// TIA Portal project "COUNTER_1_3" (V14)

(* hardware
DEVICE "S7-1200 station_1"  S7-1200 Station
   slot 0: "Rack_0"  S7-1200 Rack  Rack  V1.0
   slot 1: "CPU"  CPU 1212C DC/DC/DC  6ES7 212-1AE40-0XB0  V4.2
DEVICE "HMI_1"  KTP400 Basic PN
   slot 0: "KTP400 Basic PN"  KTP400 Basic PN  6AV2 123-2DB03-0AX0  14.0.1.0
   slot 1: "HMI_RT_1"  KTP400 Basic PN  6AV2 123-2DB03-0AX0  14.0.1.0
   slot 5: "HMI_1.IE_CP_1"  PROFINET Interface  14.0.1.0
      slot 1: "PROFINET Interface_1"  PROFINET Interface
         slot 1: "Port_1"  Port
DEVICE "HMI_2"  KTP400 Basic PN
   slot 0: "KTP400 Basic PN"  KTP400 Basic PN  6AV2 123-2DB03-0AX0  14.0.1.0
   slot 1: "HMI_RT_2"  KTP400 Basic PN  6AV2 123-2DB03-0AX0  14.0.1.0
   slot 5: "HMI_1.IE_CP_1"  PROFINET Interface  14.0.1.0
      slot 1: "PROFINET Interface_1"  PROFINET Interface
         slot 1: "Port_1"  Port
*)

// ===== PLC "CPU"  CPU 1212C DC/DC/DC =====

VAR_GLOBAL   // PLC tag table "Default tag table"
   "CNT_1_IMP" AT %ID1000 : DWord;
   "CNT_2_IMP" AT %ID1004 : DInt;
   "StopFromCNT_2" AT %Q0.0 : Bool;   // Стоп от счетчика метража машина 1
   "CNN_3_IMP" AT %ID1008 : DInt;
   "CNT_4_IMP" AT %ID1012 : DInt;
   "StopFromCNT_4" AT %Q0.1 : Bool;
   "Tag_1" AT %MW10 : Word;
   "Tag_2" AT %MD10 : Real;
   "Tag_3" AT %MD15 : Real;
END_VAR

DATA_BLOCK "DSE_1"   // DB3
{ S7_Optimized_Access := 'TRUE' }
VERSION : 0.1
   VAR RETAIN
      "Счетчик импульсов 1" : DInt;
      "Счетчик импульсов 2" : DInt;
   END_VAR
   VAR
      "Сброс счетчика 1" : Bool;
      "Сброс счетчика 2" : Bool;
   END_VAR
   VAR RETAIN
      "Диаметр колеса пасма" : Real := 0.106;
      "Количество импулсов на оборот пасма" : Real := 1.0;
      "Коэффициент счетчика пасма" : Real := 1.0;
      "Метраж пасма" : Real;
      "Коэффициент трансмиссии рамки" : Real := 1.0;
      "Шаг скрутки в метрах (выбранной ступени)" : Real;
      "Коэффициент метража жилы (выбранной ступени)" : Real := 1.0;
      "метраж жила" : Real;
      "Номер ступени" : Int;
      "Ступень 0 Шаг" : Real := 0.0091;
      "Ступень 1 Шаг" : Real := 0.0114;
      "Ступень 2 Шаг" : Real := 0.0141;
      "Ступень 3 Шаг" : Real := 0.0181;
      "Ступень 4 Шаг" : Real := 0.0228;
      "Ступень 5 Шаг" : Real := 0.0316;
      "Ступень 6 Шаг" : Real := 0.04;
      "Ступень 7 Шаг" : Real := 0.0511;
      "Ступень 8 Шаг" : Real := 0.0631;
      "Ступень 9 Шаг" : Real := 0.0794;
      "Ступень 10 Шаг" : Real := 0.091;
      "Метраж заданый" : Real;
      "Ступень 0 Коэффициент метража жилы" : Real := 0.9791;
      "Ступень 1 Коэффициент метража жилы" : Real := 0.9791;
      "Ступень 2 Коэффициент метража жилы" : Real := 0.9791;
      "Ступень 3 Коэффициент метража жилы" : Real := 0.9791;
      "Ступень 4 Коэффициент метража жилы" : Real := 0.9791;
      "Ступень 5 Коэффициент метража жилы" : Real := 0.9791;
      "Ступень 6 Коэффициент метража жилы" : Real := 0.9791;
      "Ступень 7 Коэффициент метража жилы" : Real := 0.9791;
      "Ступень 8 Коэффициент метража жилы" : Real := 0.9791;
      "Ступень 9 Коэффициент метража жилы" : Real := 0.9791;
      "Ступень 10 Коэффициент метража жилы" : Real := 0.9791;
   END_VAR
   VAR
      "Скорость DSE 1" : Real;
   END_VAR
BEGIN
END_DATA_BLOCK

DATA_BLOCK "DSE_3"   // DB6
{ S7_Optimized_Access := 'TRUE' }
VERSION : 0.1
   VAR RETAIN
      "Счетчик импульсов 1" : DInt;
      "Счетчик импульсов 2" : DInt;
   END_VAR
   VAR
      "Сброс счетчика 1" : Bool;
      "Сброс счетчика 2" : Bool;
   END_VAR
   VAR RETAIN
      "Диаметр колеса пасма" : Real := 0.106;
      "Количество импулсов на оборот пасма" : Real := 1.0;
      "Коэффициент счетчика пасма" : Real := 1.0;
      "Метраж пасма" : Real;
      "Коэффициент трансмиссии рамки" : Real := 1.0;
      "Шаг скрутки в метрах (выбранной ступени)" : Real;
      "Коэффициент метража жилы (выбранной ступени)" : Real := 1.0;
      "метраж жила" : Real;
      "Номер ступени" : Int;
      "Ступень 0 Шаг" : Real := 0.0091;
      "Ступень 1 Шаг" : Real := 0.0114;
      "Ступень 2 Шаг" : Real := 0.0141;
      "Ступень 3 Шаг" : Real := 0.0181;
      "Ступень 4 Шаг" : Real := 0.0228;
      "Ступень 5 Шаг" : Real := 0.0316;
      "Ступень 6 Шаг" : Real := 0.04;
      "Ступень 7 Шаг" : Real := 0.0511;
      "Ступень 8 Шаг" : Real := 0.0631;
      "Ступень 9 Шаг" : Real := 0.0794;
      "Ступень 10 Шаг" : Real := 0.091;
      "Метраж заданый" : Real;
      "Ступень 0 Коэффициент метража жилы" : Real := 0.9791;
      "Ступень 1 Коэффициент метража жилы" : Real := 0.9791;
      "Ступень 2 Коэффициент метража жилы" : Real := 0.9791;
      "Ступень 3 Коэффициент метража жилы" : Real := 0.9791;
      "Ступень 4 Коэффициент метража жилы" : Real := 0.9791;
      "Ступень 5 Коэффициент метража жилы" : Real := 0.9791;
      "Ступень 6 Коэффициент метража жилы" : Real := 0.9791;
      "Ступень 7 Коэффициент метража жилы" : Real := 0.9791;
      "Ступень 8 Коэффициент метража жилы" : Real := 0.9791;
      "Ступень 9 Коэффициент метража жилы" : Real := 0.9791;
      "Ступень 10 Коэффициент метража жилы" : Real := 0.9791;
   END_VAR
   VAR
      "Скорость DSE 1" : Real;
   END_VAR
BEGIN
END_DATA_BLOCK

ORGANIZATION_BLOCK "Main"   // OB1, LAD, ProgramCycle
TITLE = "Main Program Sweep (Cycle)"
{ S7_Optimized_Access := 'TRUE' }
VERSION : 0.1
   VAR_INPUT
      Initial_Call : Bool;   // Initial call of this OB
      Remanence : Bool;   // =True, if remanent data are available
   END_VAR
BEGIN

REGION Network 1: DSE 1
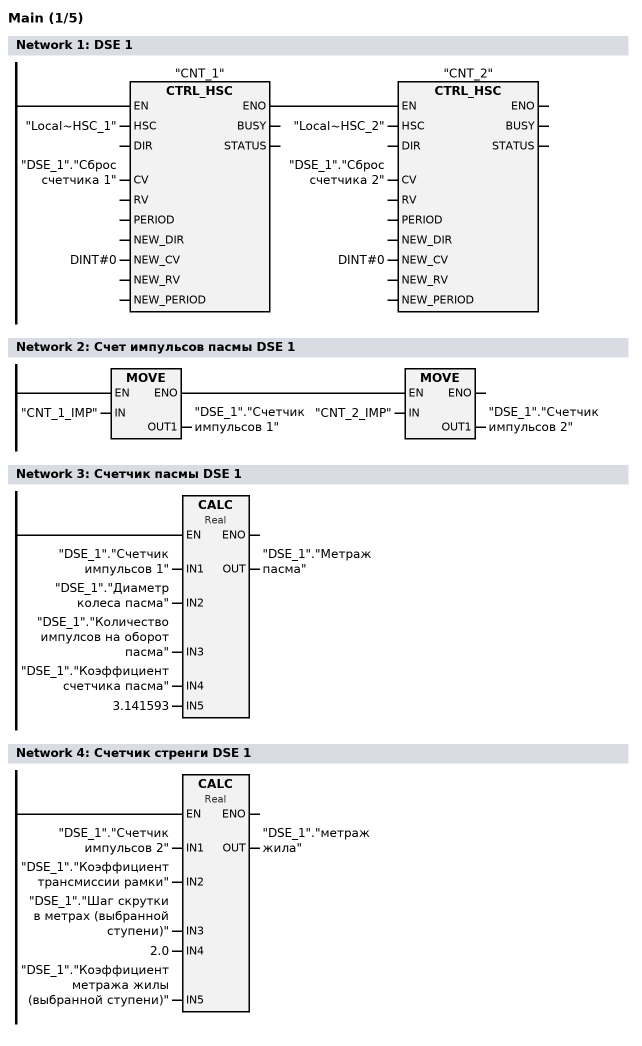
   // ENO of a box is taken as its EN; it also drops when the box reports an error
   "CNT_1"(HSC := "Local~HSC_1", CV := "DSE_1"."Сброс счетчика 1", NEW_CV := DINT#0);   // CTRL_HSC
   "CNT_2"(HSC := "Local~HSC_2", CV := "DSE_1"."Сброс счетчика 2", NEW_CV := DINT#0);   // CTRL_HSC
END_REGION

REGION Network 2: Счет импульсов пасмы DSE 1
   RUNG wire#powerrail
      Move(in := "CNT_1_IMP", out1 => "DSE_1"."Счетчик импульсов 1")
      Move(in := "CNT_2_IMP", out1 => "DSE_1"."Счетчик импульсов 2")
   END_RUNG
   // the same network as SCL:
   "DSE_1"."Счетчик импульсов 1" := "CNT_1_IMP";
   "DSE_1"."Счетчик импульсов 2" := "CNT_2_IMP";
END_REGION

REGION Network 3: Счетчик пасмы DSE 1
   CALC(in1 := "DSE_1"."Счетчик импульсов 1",
        in2 := "DSE_1"."Диаметр колеса пасма",
        in3 := "DSE_1"."Количество импулсов на оборот пасма",
        in4 := "DSE_1"."Коэффициент счетчика пасма",
        in5 := 3.141593,
        out => "DSE_1"."Метраж пасма");
END_REGION

REGION Network 4: Счетчик стренги DSE 1
   CALC(in1 := "DSE_1"."Счетчик импульсов 2",
        in2 := "DSE_1"."Коэффициент трансмиссии рамки",
        in3 := "DSE_1"."Шаг скрутки в метрах (выбранной ступени)",
        in4 := 2.0,
        in5 := "DSE_1"."Коэффициент метража жилы (выбранной ступени)",
        out => "DSE_1"."метраж жила");
END_REGION

REGION Network 5: Загрузка шага скрутки в метрах DSE 1
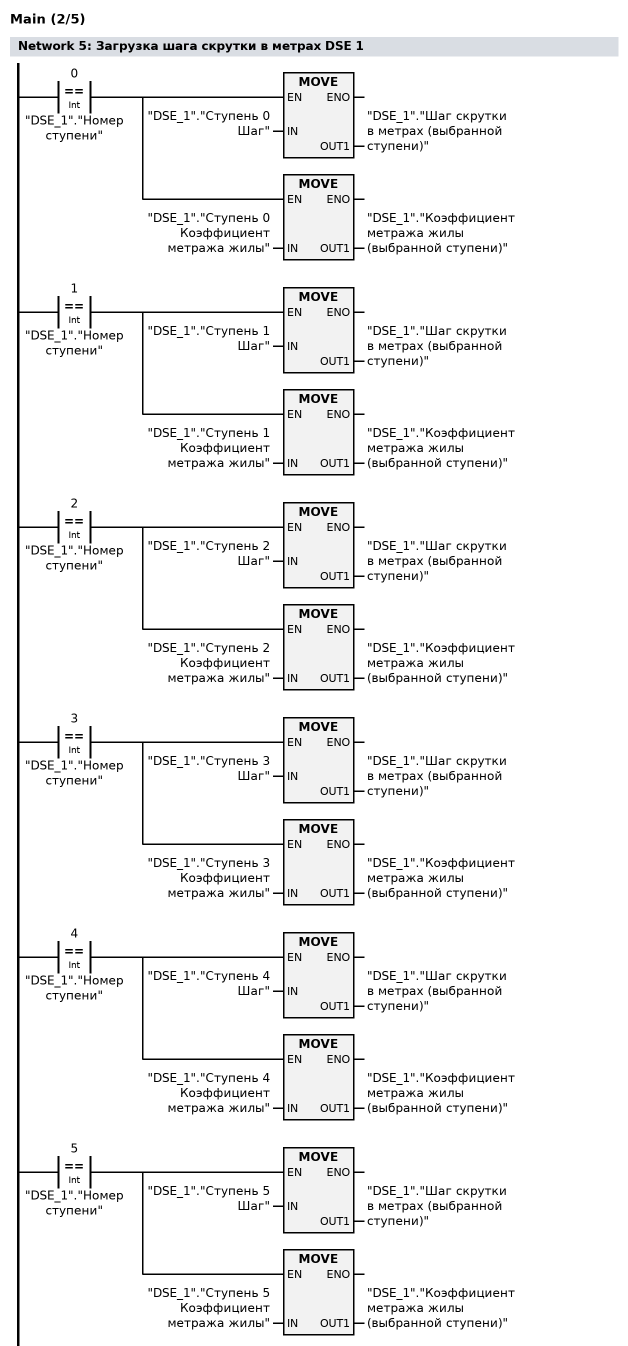
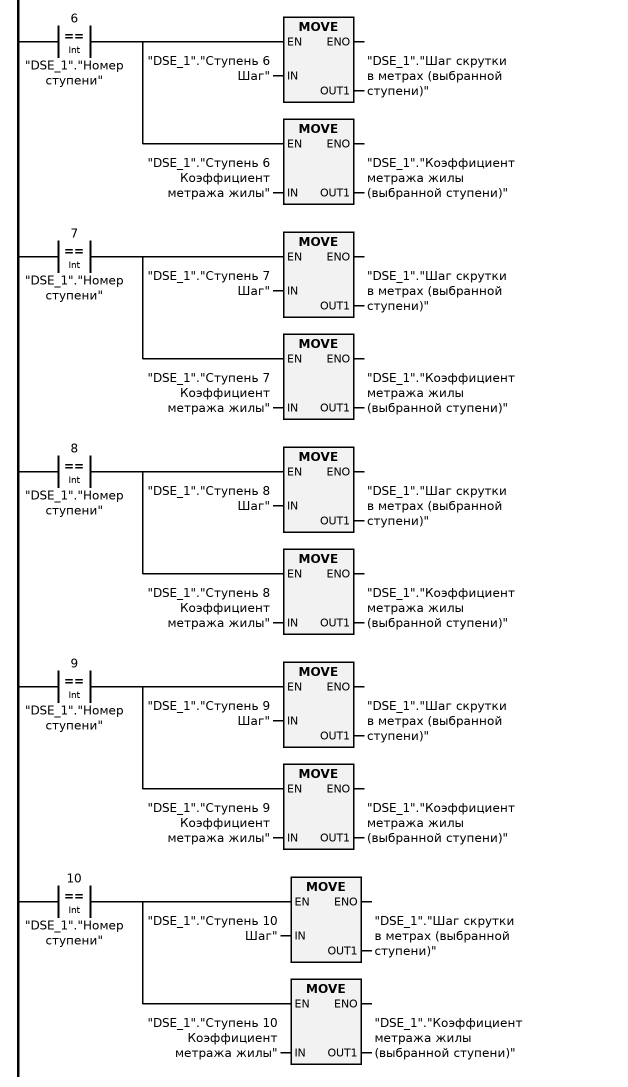
   RUNG wire#powerrail
      { S7_Templates := "SrcType := Int" } EQ_Contact(in1 := 0, in2 := "DSE_1"."Номер ступени")
      wire#w1
      Move(in := "DSE_1"."Ступень 0 Шаг", out1 => "DSE_1"."Шаг скрутки в метрах (выбранной ступени)")
   END_RUNG
   RUNG wire#w1
      Move(in := "DSE_1"."Ступень 0 Коэффициент метража жилы", out1 => "DSE_1"."Коэффициент метража жилы (выбранной ступени)")
   END_RUNG
   RUNG wire#powerrail
      { S7_Templates := "SrcType := Int" } EQ_Contact(in1 := 1, in2 := "DSE_1"."Номер ступени")
      wire#w2
      Move(in := "DSE_1"."Ступень 1 Шаг", out1 => "DSE_1"."Шаг скрутки в метрах (выбранной ступени)")
   END_RUNG
   RUNG wire#w2
      Move(in := "DSE_1"."Ступень 1 Коэффициент метража жилы", out1 => "DSE_1"."Коэффициент метража жилы (выбранной ступени)")
   END_RUNG
   RUNG wire#powerrail
      { S7_Templates := "SrcType := Int" } EQ_Contact(in1 := 2, in2 := "DSE_1"."Номер ступени")
      wire#w3
      Move(in := "DSE_1"."Ступень 2 Шаг", out1 => "DSE_1"."Шаг скрутки в метрах (выбранной ступени)")
   END_RUNG
   RUNG wire#w3
      Move(in := "DSE_1"."Ступень 2 Коэффициент метража жилы", out1 => "DSE_1"."Коэффициент метража жилы (выбранной ступени)")
   END_RUNG
   RUNG wire#powerrail
      { S7_Templates := "SrcType := Int" } EQ_Contact(in1 := 3, in2 := "DSE_1"."Номер ступени")
      wire#w4
      Move(in := "DSE_1"."Ступень 3 Шаг", out1 => "DSE_1"."Шаг скрутки в метрах (выбранной ступени)")
   END_RUNG
   RUNG wire#w4
      Move(in := "DSE_1"."Ступень 3 Коэффициент метража жилы", out1 => "DSE_1"."Коэффициент метража жилы (выбранной ступени)")
   END_RUNG
   RUNG wire#powerrail
      { S7_Templates := "SrcType := Int" } EQ_Contact(in1 := 4, in2 := "DSE_1"."Номер ступени")
      wire#w5
      Move(in := "DSE_1"."Ступень 4 Шаг", out1 => "DSE_1"."Шаг скрутки в метрах (выбранной ступени)")
   END_RUNG
   RUNG wire#w5
      Move(in := "DSE_1"."Ступень 4 Коэффициент метража жилы", out1 => "DSE_1"."Коэффициент метража жилы (выбранной ступени)")
   END_RUNG
   RUNG wire#powerrail
      { S7_Templates := "SrcType := Int" } EQ_Contact(in1 := 5, in2 := "DSE_1"."Номер ступени")
      wire#w6
      Move(in := "DSE_1"."Ступень 5 Шаг", out1 => "DSE_1"."Шаг скрутки в метрах (выбранной ступени)")
   END_RUNG
   RUNG wire#w6
      Move(in := "DSE_1"."Ступень 5 Коэффициент метража жилы", out1 => "DSE_1"."Коэффициент метража жилы (выбранной ступени)")
   END_RUNG
   RUNG wire#powerrail
      { S7_Templates := "SrcType := Int" } EQ_Contact(in1 := 6, in2 := "DSE_1"."Номер ступени")
      wire#w7
      Move(in := "DSE_1"."Ступень 6 Шаг", out1 => "DSE_1"."Шаг скрутки в метрах (выбранной ступени)")
   END_RUNG
   RUNG wire#w7
      Move(in := "DSE_1"."Ступень 6 Коэффициент метража жилы", out1 => "DSE_1"."Коэффициент метража жилы (выбранной ступени)")
   END_RUNG
   RUNG wire#powerrail
      { S7_Templates := "SrcType := Int" } EQ_Contact(in1 := 7, in2 := "DSE_1"."Номер ступени")
      wire#w8
      Move(in := "DSE_1"."Ступень 7 Шаг", out1 => "DSE_1"."Шаг скрутки в метрах (выбранной ступени)")
   END_RUNG
   RUNG wire#w8
      Move(in := "DSE_1"."Ступень 7 Коэффициент метража жилы", out1 => "DSE_1"."Коэффициент метража жилы (выбранной ступени)")
   END_RUNG
   RUNG wire#powerrail
      { S7_Templates := "SrcType := Int" } EQ_Contact(in1 := 8, in2 := "DSE_1"."Номер ступени")
      wire#w9
      Move(in := "DSE_1"."Ступень 8 Шаг", out1 => "DSE_1"."Шаг скрутки в метрах (выбранной ступени)")
   END_RUNG
   RUNG wire#w9
      Move(in := "DSE_1"."Ступень 8 Коэффициент метража жилы", out1 => "DSE_1"."Коэффициент метража жилы (выбранной ступени)")
   END_RUNG
   RUNG wire#powerrail
      { S7_Templates := "SrcType := Int" } EQ_Contact(in1 := 9, in2 := "DSE_1"."Номер ступени")
      wire#w10
      Move(in := "DSE_1"."Ступень 9 Шаг", out1 => "DSE_1"."Шаг скрутки в метрах (выбранной ступени)")
   END_RUNG
   RUNG wire#w10
      Move(in := "DSE_1"."Ступень 9 Коэффициент метража жилы", out1 => "DSE_1"."Коэффициент метража жилы (выбранной ступени)")
   END_RUNG
   RUNG wire#powerrail
      { S7_Templates := "SrcType := Int" } EQ_Contact(in1 := 10, in2 := "DSE_1"."Номер ступени")
      wire#w11
      Move(in := "DSE_1"."Ступень 10 Шаг", out1 => "DSE_1"."Шаг скрутки в метрах (выбранной ступени)")
   END_RUNG
   RUNG wire#w11
      Move(in := "DSE_1"."Ступень 10 Коэффициент метража жилы", out1 => "DSE_1"."Коэффициент метража жилы (выбранной ступени)")
   END_RUNG
   // the same network as SCL:
   IF 0 = "DSE_1"."Номер ступени" THEN
       "DSE_1"."Шаг скрутки в метрах (выбранной ступени)" := "DSE_1"."Ступень 0 Шаг";
       "DSE_1"."Коэффициент метража жилы (выбранной ступени)" := "DSE_1"."Ступень 0 Коэффициент метража жилы";
   END_IF;
   IF 1 = "DSE_1"."Номер ступени" THEN
       "DSE_1"."Шаг скрутки в метрах (выбранной ступени)" := "DSE_1"."Ступень 1 Шаг";
       "DSE_1"."Коэффициент метража жилы (выбранной ступени)" := "DSE_1"."Ступень 1 Коэффициент метража жилы";
   END_IF;
   IF 2 = "DSE_1"."Номер ступени" THEN
       "DSE_1"."Шаг скрутки в метрах (выбранной ступени)" := "DSE_1"."Ступень 2 Шаг";
       "DSE_1"."Коэффициент метража жилы (выбранной ступени)" := "DSE_1"."Ступень 2 Коэффициент метража жилы";
   END_IF;
   IF 3 = "DSE_1"."Номер ступени" THEN
       "DSE_1"."Шаг скрутки в метрах (выбранной ступени)" := "DSE_1"."Ступень 3 Шаг";
       "DSE_1"."Коэффициент метража жилы (выбранной ступени)" := "DSE_1"."Ступень 3 Коэффициент метража жилы";
   END_IF;
   IF 4 = "DSE_1"."Номер ступени" THEN
       "DSE_1"."Шаг скрутки в метрах (выбранной ступени)" := "DSE_1"."Ступень 4 Шаг";
       "DSE_1"."Коэффициент метража жилы (выбранной ступени)" := "DSE_1"."Ступень 4 Коэффициент метража жилы";
   END_IF;
   IF 5 = "DSE_1"."Номер ступени" THEN
       "DSE_1"."Шаг скрутки в метрах (выбранной ступени)" := "DSE_1"."Ступень 5 Шаг";
       "DSE_1"."Коэффициент метража жилы (выбранной ступени)" := "DSE_1"."Ступень 5 Коэффициент метража жилы";
   END_IF;
   IF 6 = "DSE_1"."Номер ступени" THEN
       "DSE_1"."Шаг скрутки в метрах (выбранной ступени)" := "DSE_1"."Ступень 6 Шаг";
       "DSE_1"."Коэффициент метража жилы (выбранной ступени)" := "DSE_1"."Ступень 6 Коэффициент метража жилы";
   END_IF;
   IF 7 = "DSE_1"."Номер ступени" THEN
       "DSE_1"."Шаг скрутки в метрах (выбранной ступени)" := "DSE_1"."Ступень 7 Шаг";
       "DSE_1"."Коэффициент метража жилы (выбранной ступени)" := "DSE_1"."Ступень 7 Коэффициент метража жилы";
   END_IF;
   IF 8 = "DSE_1"."Номер ступени" THEN
       "DSE_1"."Шаг скрутки в метрах (выбранной ступени)" := "DSE_1"."Ступень 8 Шаг";
       "DSE_1"."Коэффициент метража жилы (выбранной ступени)" := "DSE_1"."Ступень 8 Коэффициент метража жилы";
   END_IF;
   IF 9 = "DSE_1"."Номер ступени" THEN
       "DSE_1"."Шаг скрутки в метрах (выбранной ступени)" := "DSE_1"."Ступень 9 Шаг";
       "DSE_1"."Коэффициент метража жилы (выбранной ступени)" := "DSE_1"."Ступень 9 Коэффициент метража жилы";
   END_IF;
   IF 10 = "DSE_1"."Номер ступени" THEN
       "DSE_1"."Шаг скрутки в метрах (выбранной ступени)" := "DSE_1"."Ступень 10 Шаг";
       "DSE_1"."Коэффициент метража жилы (выбранной ступени)" := "DSE_1"."Ступень 10 Коэффициент метража жилы";
   END_IF;
END_REGION

REGION Network 6: Стоп по счетчику DSE 1
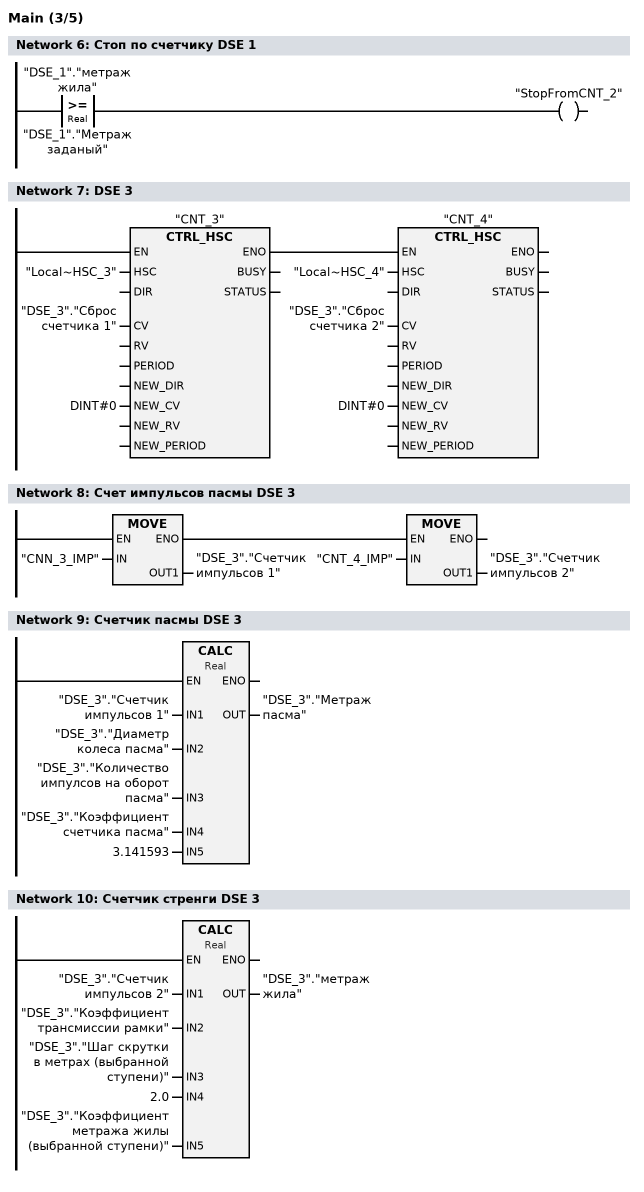
   RUNG wire#powerrail
      { S7_Templates := "SrcType := Real" } GE_Contact(in1 := "DSE_1"."метраж жила", in2 := "DSE_1"."Метраж заданый")
      Coil( "StopFromCNT_2" )
   END_RUNG
   // the same network as SCL:
   "StopFromCNT_2" := "DSE_1"."метраж жила" >= "DSE_1"."Метраж заданый";
END_REGION

REGION Network 7: DSE 3
   // ENO of a box is taken as its EN; it also drops when the box reports an error
   "CNT_3"(HSC := "Local~HSC_3", CV := "DSE_3"."Сброс счетчика 1", NEW_CV := DINT#0);   // CTRL_HSC
   "CNT_4"(HSC := "Local~HSC_4", CV := "DSE_3"."Сброс счетчика 2", NEW_CV := DINT#0);   // CTRL_HSC
END_REGION

REGION Network 8: Счет импульсов пасмы DSE 3
   RUNG wire#powerrail
      Move(in := "CNN_3_IMP", out1 => "DSE_3"."Счетчик импульсов 1")
      Move(in := "CNT_4_IMP", out1 => "DSE_3"."Счетчик импульсов 2")
   END_RUNG
   // the same network as SCL:
   "DSE_3"."Счетчик импульсов 1" := "CNN_3_IMP";
   "DSE_3"."Счетчик импульсов 2" := "CNT_4_IMP";
END_REGION

REGION Network 9: Счетчик пасмы DSE 3
   CALC(in1 := "DSE_3"."Счетчик импульсов 1",
        in2 := "DSE_3"."Диаметр колеса пасма",
        in3 := "DSE_3"."Количество импулсов на оборот пасма",
        in4 := "DSE_3"."Коэффициент счетчика пасма",
        in5 := 3.141593,
        out => "DSE_3"."Метраж пасма");
END_REGION

REGION Network 10: Счетчик стренги DSE 3
   CALC(in1 := "DSE_3"."Счетчик импульсов 2",
        in2 := "DSE_3"."Коэффициент трансмиссии рамки",
        in3 := "DSE_3"."Шаг скрутки в метрах (выбранной ступени)",
        in4 := 2.0,
        in5 := "DSE_3"."Коэффициент метража жилы (выбранной ступени)",
        out => "DSE_3"."метраж жила");
END_REGION

REGION Network 11: Загрузка шага скрутки в метрах DSE 3
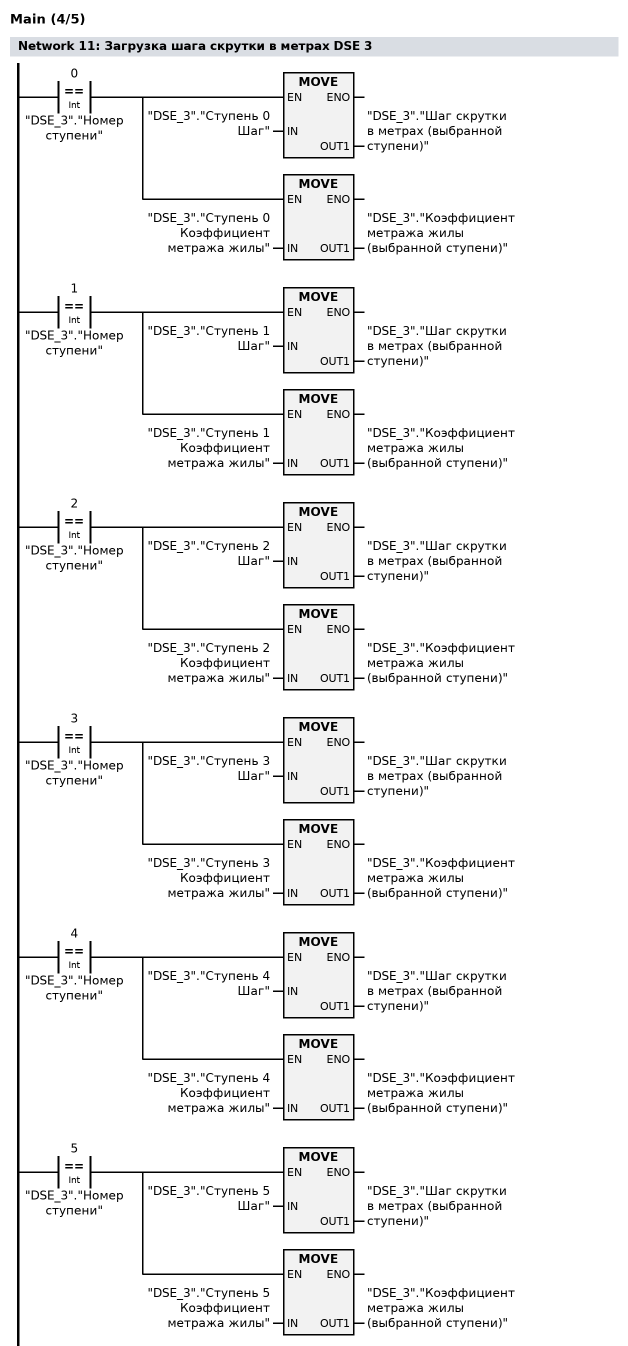
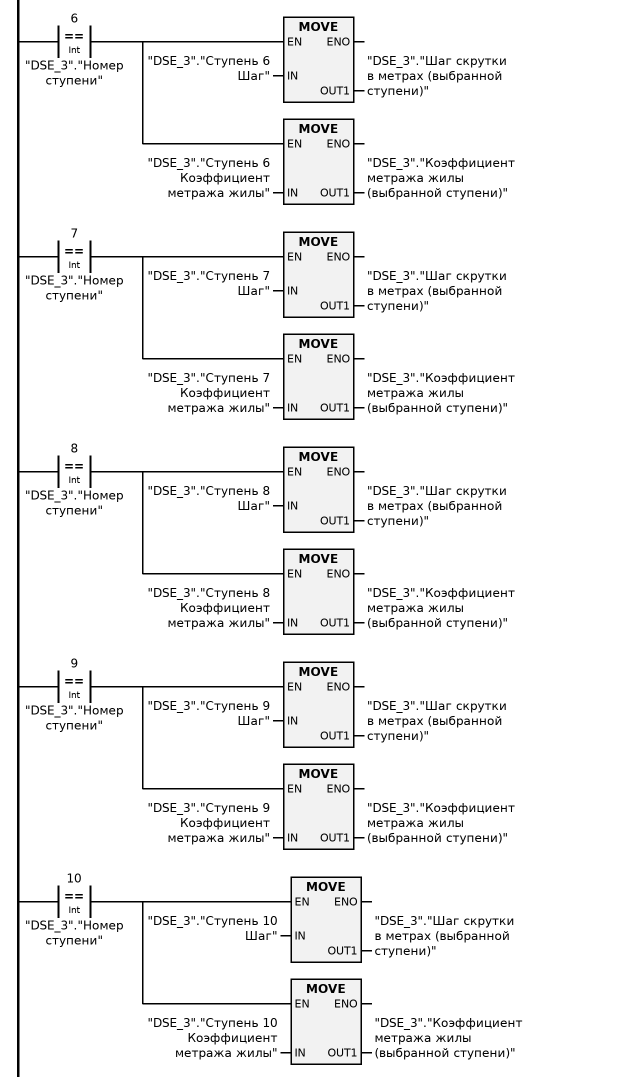
   RUNG wire#powerrail
      { S7_Templates := "SrcType := Int" } EQ_Contact(in1 := 0, in2 := "DSE_3"."Номер ступени")
      wire#w1
      Move(in := "DSE_3"."Ступень 0 Шаг", out1 => "DSE_3"."Шаг скрутки в метрах (выбранной ступени)")
   END_RUNG
   RUNG wire#w1
      Move(in := "DSE_3"."Ступень 0 Коэффициент метража жилы", out1 => "DSE_3"."Коэффициент метража жилы (выбранной ступени)")
   END_RUNG
   RUNG wire#powerrail
      { S7_Templates := "SrcType := Int" } EQ_Contact(in1 := 1, in2 := "DSE_3"."Номер ступени")
      wire#w2
      Move(in := "DSE_3"."Ступень 1 Шаг", out1 => "DSE_3"."Шаг скрутки в метрах (выбранной ступени)")
   END_RUNG
   RUNG wire#w2
      Move(in := "DSE_3"."Ступень 1 Коэффициент метража жилы", out1 => "DSE_3"."Коэффициент метража жилы (выбранной ступени)")
   END_RUNG
   RUNG wire#powerrail
      { S7_Templates := "SrcType := Int" } EQ_Contact(in1 := 2, in2 := "DSE_3"."Номер ступени")
      wire#w3
      Move(in := "DSE_3"."Ступень 2 Шаг", out1 => "DSE_3"."Шаг скрутки в метрах (выбранной ступени)")
   END_RUNG
   RUNG wire#w3
      Move(in := "DSE_3"."Ступень 2 Коэффициент метража жилы", out1 => "DSE_3"."Коэффициент метража жилы (выбранной ступени)")
   END_RUNG
   RUNG wire#powerrail
      { S7_Templates := "SrcType := Int" } EQ_Contact(in1 := 3, in2 := "DSE_3"."Номер ступени")
      wire#w4
      Move(in := "DSE_3"."Ступень 3 Шаг", out1 => "DSE_3"."Шаг скрутки в метрах (выбранной ступени)")
   END_RUNG
   RUNG wire#w4
      Move(in := "DSE_3"."Ступень 3 Коэффициент метража жилы", out1 => "DSE_3"."Коэффициент метража жилы (выбранной ступени)")
   END_RUNG
   RUNG wire#powerrail
      { S7_Templates := "SrcType := Int" } EQ_Contact(in1 := 4, in2 := "DSE_3"."Номер ступени")
      wire#w5
      Move(in := "DSE_3"."Ступень 4 Шаг", out1 => "DSE_3"."Шаг скрутки в метрах (выбранной ступени)")
   END_RUNG
   RUNG wire#w5
      Move(in := "DSE_3"."Ступень 4 Коэффициент метража жилы", out1 => "DSE_3"."Коэффициент метража жилы (выбранной ступени)")
   END_RUNG
   RUNG wire#powerrail
      { S7_Templates := "SrcType := Int" } EQ_Contact(in1 := 5, in2 := "DSE_3"."Номер ступени")
      wire#w6
      Move(in := "DSE_3"."Ступень 5 Шаг", out1 => "DSE_3"."Шаг скрутки в метрах (выбранной ступени)")
   END_RUNG
   RUNG wire#w6
      Move(in := "DSE_3"."Ступень 5 Коэффициент метража жилы", out1 => "DSE_3"."Коэффициент метража жилы (выбранной ступени)")
   END_RUNG
   RUNG wire#powerrail
      { S7_Templates := "SrcType := Int" } EQ_Contact(in1 := 6, in2 := "DSE_3"."Номер ступени")
      wire#w7
      Move(in := "DSE_3"."Ступень 6 Шаг", out1 => "DSE_3"."Шаг скрутки в метрах (выбранной ступени)")
   END_RUNG
   RUNG wire#w7
      Move(in := "DSE_3"."Ступень 6 Коэффициент метража жилы", out1 => "DSE_3"."Коэффициент метража жилы (выбранной ступени)")
   END_RUNG
   RUNG wire#powerrail
      { S7_Templates := "SrcType := Int" } EQ_Contact(in1 := 7, in2 := "DSE_3"."Номер ступени")
      wire#w8
      Move(in := "DSE_3"."Ступень 7 Шаг", out1 => "DSE_3"."Шаг скрутки в метрах (выбранной ступени)")
   END_RUNG
   RUNG wire#w8
      Move(in := "DSE_3"."Ступень 7 Коэффициент метража жилы", out1 => "DSE_3"."Коэффициент метража жилы (выбранной ступени)")
   END_RUNG
   RUNG wire#powerrail
      { S7_Templates := "SrcType := Int" } EQ_Contact(in1 := 8, in2 := "DSE_3"."Номер ступени")
      wire#w9
      Move(in := "DSE_3"."Ступень 8 Шаг", out1 => "DSE_3"."Шаг скрутки в метрах (выбранной ступени)")
   END_RUNG
   RUNG wire#w9
      Move(in := "DSE_3"."Ступень 8 Коэффициент метража жилы", out1 => "DSE_3"."Коэффициент метража жилы (выбранной ступени)")
   END_RUNG
   RUNG wire#powerrail
      { S7_Templates := "SrcType := Int" } EQ_Contact(in1 := 9, in2 := "DSE_3"."Номер ступени")
      wire#w10
      Move(in := "DSE_3"."Ступень 9 Шаг", out1 => "DSE_3"."Шаг скрутки в метрах (выбранной ступени)")
   END_RUNG
   RUNG wire#w10
      Move(in := "DSE_3"."Ступень 9 Коэффициент метража жилы", out1 => "DSE_3"."Коэффициент метража жилы (выбранной ступени)")
   END_RUNG
   RUNG wire#powerrail
      { S7_Templates := "SrcType := Int" } EQ_Contact(in1 := 10, in2 := "DSE_3"."Номер ступени")
      wire#w11
      Move(in := "DSE_3"."Ступень 10 Шаг", out1 => "DSE_3"."Шаг скрутки в метрах (выбранной ступени)")
   END_RUNG
   RUNG wire#w11
      Move(in := "DSE_3"."Ступень 10 Коэффициент метража жилы", out1 => "DSE_3"."Коэффициент метража жилы (выбранной ступени)")
   END_RUNG
   // the same network as SCL:
   IF 0 = "DSE_3"."Номер ступени" THEN
       "DSE_3"."Шаг скрутки в метрах (выбранной ступени)" := "DSE_3"."Ступень 0 Шаг";
       "DSE_3"."Коэффициент метража жилы (выбранной ступени)" := "DSE_3"."Ступень 0 Коэффициент метража жилы";
   END_IF;
   IF 1 = "DSE_3"."Номер ступени" THEN
       "DSE_3"."Шаг скрутки в метрах (выбранной ступени)" := "DSE_3"."Ступень 1 Шаг";
       "DSE_3"."Коэффициент метража жилы (выбранной ступени)" := "DSE_3"."Ступень 1 Коэффициент метража жилы";
   END_IF;
   IF 2 = "DSE_3"."Номер ступени" THEN
       "DSE_3"."Шаг скрутки в метрах (выбранной ступени)" := "DSE_3"."Ступень 2 Шаг";
       "DSE_3"."Коэффициент метража жилы (выбранной ступени)" := "DSE_3"."Ступень 2 Коэффициент метража жилы";
   END_IF;
   IF 3 = "DSE_3"."Номер ступени" THEN
       "DSE_3"."Шаг скрутки в метрах (выбранной ступени)" := "DSE_3"."Ступень 3 Шаг";
       "DSE_3"."Коэффициент метража жилы (выбранной ступени)" := "DSE_3"."Ступень 3 Коэффициент метража жилы";
   END_IF;
   IF 4 = "DSE_3"."Номер ступени" THEN
       "DSE_3"."Шаг скрутки в метрах (выбранной ступени)" := "DSE_3"."Ступень 4 Шаг";
       "DSE_3"."Коэффициент метража жилы (выбранной ступени)" := "DSE_3"."Ступень 4 Коэффициент метража жилы";
   END_IF;
   IF 5 = "DSE_3"."Номер ступени" THEN
       "DSE_3"."Шаг скрутки в метрах (выбранной ступени)" := "DSE_3"."Ступень 5 Шаг";
       "DSE_3"."Коэффициент метража жилы (выбранной ступени)" := "DSE_3"."Ступень 5 Коэффициент метража жилы";
   END_IF;
   IF 6 = "DSE_3"."Номер ступени" THEN
       "DSE_3"."Шаг скрутки в метрах (выбранной ступени)" := "DSE_3"."Ступень 6 Шаг";
       "DSE_3"."Коэффициент метража жилы (выбранной ступени)" := "DSE_3"."Ступень 6 Коэффициент метража жилы";
   END_IF;
   IF 7 = "DSE_3"."Номер ступени" THEN
       "DSE_3"."Шаг скрутки в метрах (выбранной ступени)" := "DSE_3"."Ступень 7 Шаг";
       "DSE_3"."Коэффициент метража жилы (выбранной ступени)" := "DSE_3"."Ступень 7 Коэффициент метража жилы";
   END_IF;
   IF 8 = "DSE_3"."Номер ступени" THEN
       "DSE_3"."Шаг скрутки в метрах (выбранной ступени)" := "DSE_3"."Ступень 8 Шаг";
       "DSE_3"."Коэффициент метража жилы (выбранной ступени)" := "DSE_3"."Ступень 8 Коэффициент метража жилы";
   END_IF;
   IF 9 = "DSE_3"."Номер ступени" THEN
       "DSE_3"."Шаг скрутки в метрах (выбранной ступени)" := "DSE_3"."Ступень 9 Шаг";
       "DSE_3"."Коэффициент метража жилы (выбранной ступени)" := "DSE_3"."Ступень 9 Коэффициент метража жилы";
   END_IF;
   IF 10 = "DSE_3"."Номер ступени" THEN
       "DSE_3"."Шаг скрутки в метрах (выбранной ступени)" := "DSE_3"."Ступень 10 Шаг";
       "DSE_3"."Коэффициент метража жилы (выбранной ступени)" := "DSE_3"."Ступень 10 Коэффициент метража жилы";
   END_IF;
END_REGION

REGION Network 12: Стоп по счетчику DSE 3
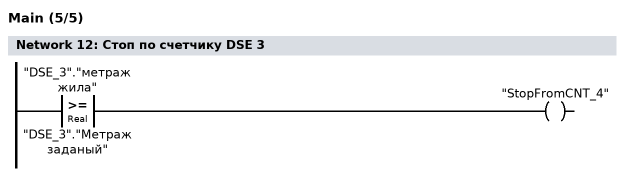
   RUNG wire#powerrail
      { S7_Templates := "SrcType := Real" } GE_Contact(in1 := "DSE_3"."метраж жила", in2 := "DSE_3"."Метраж заданый")
      Coil( "StopFromCNT_4" )
   END_RUNG
   // the same network as SCL:
   "StopFromCNT_4" := "DSE_3"."метраж жила" >= "DSE_3"."Метраж заданый";
END_REGION
END_ORGANIZATION_BLOCK

ORGANIZATION_BLOCK "Cyclic interrupt"   // OB30, LAD, CyclicInterrupt
{ S7_Optimized_Access := 'TRUE' }
VERSION : 0.1
   VAR_INPUT
      Initial_Call : Bool;   // Initial call of this OB
      Event_Count : Int;   // Events discarded
   END_VAR
BEGIN

REGION Network 1
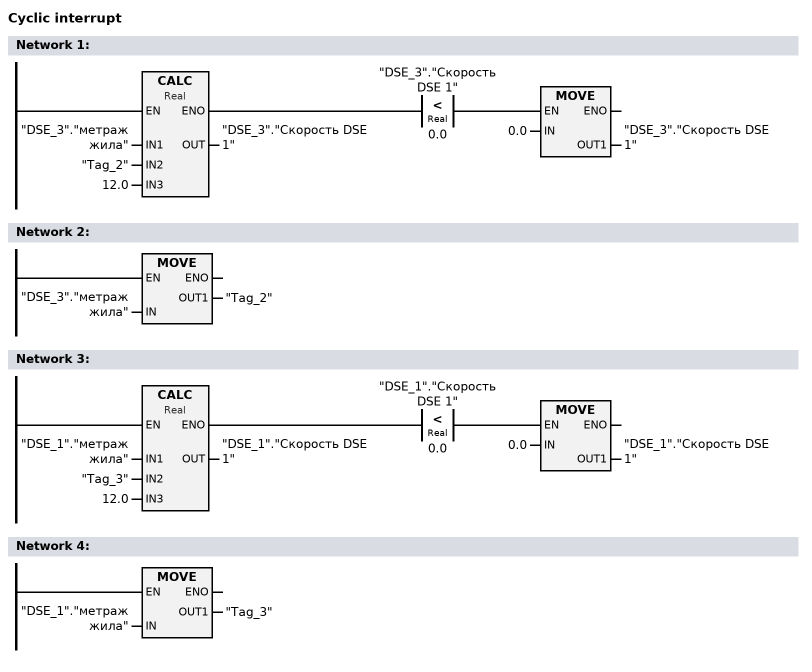
   CALC(in1 := "DSE_3"."метраж жила", in2 := "Tag_2", in3 := 12.0, out => "DSE_3"."Скорость DSE 1");
   IF "DSE_3"."Скорость DSE 1" < 0.0 THEN "DSE_3"."Скорость DSE 1" := 0.0; END_IF;
END_REGION

REGION Network 2
   RUNG wire#powerrail
      Move(in := "DSE_3"."метраж жила", out1 => "Tag_2")
   END_RUNG
   // the same network as SCL:
   "Tag_2" := "DSE_3"."метраж жила";
END_REGION

REGION Network 3
   CALC(in1 := "DSE_1"."метраж жила", in2 := "Tag_3", in3 := 12.0, out => "DSE_1"."Скорость DSE 1");
   IF "DSE_1"."Скорость DSE 1" < 0.0 THEN "DSE_1"."Скорость DSE 1" := 0.0; END_IF;
END_REGION

REGION Network 4
   RUNG wire#powerrail
      Move(in := "DSE_1"."метраж жила", out1 => "Tag_3")
   END_RUNG
   // the same network as SCL:
   "Tag_3" := "DSE_1"."метраж жила";
END_REGION
END_ORGANIZATION_BLOCK

ORGANIZATION_BLOCK "Startup"   // OB100, LAD, Startup
TITLE = "Complete Restart"
{ S7_Optimized_Access := 'TRUE' }
VERSION : 0.1
   VAR_INPUT
      LostRetentive : Bool;   // True if retentive data are lost
      LostRTC : Bool;   // True if date and time are lost
   END_VAR
BEGIN

REGION Network 1: DSE 1
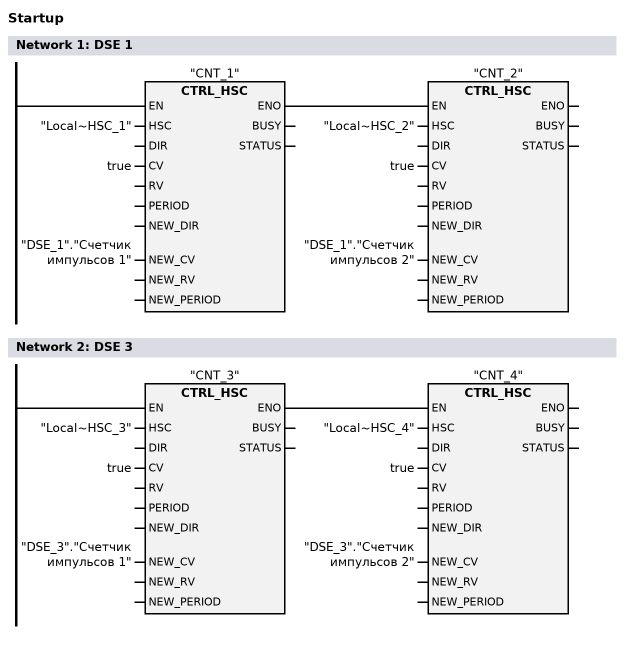
   // ENO of a box is taken as its EN; it also drops when the box reports an error
   "CNT_1"(HSC := "Local~HSC_1", CV := true, NEW_CV := "DSE_1"."Счетчик импульсов 1");   // CTRL_HSC
   "CNT_2"(HSC := "Local~HSC_2", CV := true, NEW_CV := "DSE_1"."Счетчик импульсов 2");   // CTRL_HSC
END_REGION

REGION Network 2: DSE 3
   // ENO of a box is taken as its EN; it also drops when the box reports an error
   "CNT_3"(HSC := "Local~HSC_3", CV := true, NEW_CV := "DSE_3"."Счетчик импульсов 1");   // CTRL_HSC
   "CNT_4"(HSC := "Local~HSC_4", CV := true, NEW_CV := "DSE_3"."Счетчик импульсов 2");   // CTRL_HSC
END_REGION
END_ORGANIZATION_BLOCK

(* ===== HMI "HMI_RT_1" =====
system functions are stored by id; their names below are inferred from use
connection "Connection_1": ETHERNET, SMART_S7_1200_OMS
connection "HMI_Connection_1": ETHERNET, SMART_S7_1200_OMS

HMI tags "Default tag table"
   "DSE_1_Метраж пасма" : Real = PLC DSE_1."Метраж пасма", 500 ms
   "DSE_1_метраж жила" : Real = PLC DSE_1."метраж жила", 500 ms
   "DSE_1_Шаг скрутки в метрах (выбранной ступени)" : Real = PLC DSE_1."Шаг скрутки в метрах (выбранной ступени)", 1 s
   "DSE_1_Номер ступени" : Int = PLC DSE_1."Номер ступени", 1 s
   "DSE_1_Сброс счетчика 1" : Bool = PLC DSE_1."Сброс счетчика 1", 1 s
   "DSE_1_Сброс счетчика 2" : Bool = PLC DSE_1."Сброс счетчика 2", 1 s
   "DSE_1_Диаметр колеса пасма" : Real = PLC DSE_1."Диаметр колеса пасма", 1 s
   "DSE_1_Количество импулсов на оборот пасма" : Real = PLC DSE_1."Количество импулсов на оборот пасма", 1 s
   "DSE_1_Коэффициент счетчика пасма" : Real = PLC DSE_1."Коэффициент счетчика пасма", 1 s
   "DSE_1_Коэффициент трансмиссии рамки" : Real = PLC DSE_1."Коэффициент трансмиссии рамки", 1 s
   "DSE_1_Коэффициент метража жилы (выбранной ступени)" : Real = PLC DSE_1."Коэффициент метража жилы (выбранной ступени)", 1 s
   "DSE_1_Метраж заданый" : Real = PLC DSE_1."Метраж заданый", 1 s
   "DSE_1_Ступень 0 Коэффициент метража жилы" : Real = PLC DSE_1."Ступень 0 Коэффициент метража жилы" AT %DB1.DBD0, 1 s
   "DSE_1_Ступень 1 Коэффициент метража жилы" : Real = PLC DSE_1."Ступень 1 Коэффициент метража жилы" AT %DB1.DBD0, 1 s
   "DSE_1_Ступень 2 Коэффициент метража жилы" : Real = PLC DSE_1."Ступень 2 Коэффициент метража жилы" AT %DB1.DBD0, 1 s
   "DSE_1_Ступень 3 Коэффициент метража жилы" : Real = PLC DSE_1."Ступень 3 Коэффициент метража жилы" AT %DB1.DBD0, 1 s
   "DSE_1_Ступень 4 Коэффициент метража жилы" : Real = PLC DSE_1."Ступень 4 Коэффициент метража жилы" AT %DB1.DBD0, 1 s
   "DSE_1_Ступень 5 Коэффициент метража жилы" : Real = PLC DSE_1."Ступень 5 Коэффициент метража жилы" AT %DB1.DBD0, 1 s
   "DSE_1_Ступень 6 Коэффициент метража жилы" : Real = PLC DSE_1."Ступень 6 Коэффициент метража жилы" AT %DB1.DBD0, 1 s
   "DSE_1_Ступень 7 Коэффициент метража жилы" : Real = PLC DSE_1."Ступень 7 Коэффициент метража жилы" AT %DB1.DBD0, 1 s
   "DSE_1_Ступень 8 Коэффициент метража жилы" : Real = PLC DSE_1."Ступень 8 Коэффициент метража жилы" AT %DB1.DBD0, 1 s
   "DSE_1_Ступень 9 Коэффициент метража жилы" : Real = PLC DSE_1."Ступень 9 Коэффициент метража жилы" AT %DB1.DBD0, 1 s
   "DSE_1_Скорость DSE 1" : Real = PLC DSE_1."Скорость DSE 1", 1 s
   "DSE_1_Ступень 10 Коэффициент метража жилы" : Real = PLC DSE_1."Ступень 10 Коэффициент метража жилы" AT %DB1.DBD0, 1 s

text list "Шаг_скрутки": 0 '9'; 1 '11'; 2 '14'; 3 '18'; 4 '23'; 5 '32'; 6 '40'; 7 '51'; 8 '63'; 9 '79'; 10 '91'

screen "DSE1" 480x272, template "Template_1"
   IOField "I/O field_1" at 226,233 size 111x29; FormatPattern 99999.99
      ProcessValue <- "DSE_1_Метраж пасма"
   TextField "Text field_1" at 109,233 size 109x29; Text 'пасма, м:'
   IOField "I/O field_2" at 199,74 size 255x62; FormatPattern 99999.99
      ProcessValue <- "DSE_1_метраж жила"
   TextField "Text field_2" at 7,20 size 113x37; Text 'стренга'
   SymbolicIOField "Symbolic I/O field_1" at 130,49 size 128x37; TextOff '0'; TextOn '1'; TextList "Шаг_скрутки"
      ProcessValue <- "DSE_1_Номер ступени"
   TextField "Text field_5" at 66,57 size 55x29; Text 'шаг:'
   TextField "Text field_3" at 8,97 size 149x29; Text 'намотано, м:'
   IOField "I/O field_3" at 199,174 size 174x41; FormatPattern 99999.9
      ProcessValue <- "DSE_1_Метраж заданый"
   TextField "Text field_4" at 8,179 size 182x29; Text 'установлено, м:'
   TextField "Text field_6" at 218,5 size 76x30; Text 'ДШЁ 1'
   Button "Button_1" at 27,231 size 64x41; TextOff 'сброс'
      on Press: function_b14e0dd5("DSE_1_Сброс счетчика 1", 0)
   Button "Button_2" at 384,231 size 64x41; TextOff 'сброс'
      on Press: function_b14e0dd5("DSE_1_Сброс счетчика 2", 0)
   Button "Button_3" at 433,5 size 37x30; TextOff 'Text'; PictureOff "Graphic_2"; Authorization "User administration"
      on Click: ActivateScreen("Settings", 0)
   TextField "Text field_7" at 8,138 size 188x29; Text 'скорость м/мин:'
   IOField "I/O field_4" at 199,134 size 174x41; FormatPattern 999.9
      ProcessValue <- "DSE_1_Скорость DSE 1"

screen "Settings" 480x272, template "Template_1"
   Button "Button_3" at 306,7 size 36x28; TextOff 'Text'; PictureOff "NavigateHome_KTP400_Basic_PN_TR"
      on Click: ActivateScreen("DSE1", 0)
   TextField "Text field_6" at 17,5 size 121x30; Text 'настройки'
   IOField "I/O field_1" at 35,90 size 96x32; FormatPattern 999.99
      ProcessValue <- "DSE_1_Диаметр колеса пасма"
   IOField "I/O field_2" at 35,150 size 96x32; FormatPattern 99
      ProcessValue <- "DSE_1_Количество импулсов на оборот пасма"
   IOField "I/O field_3" at 35,210 size 96x32; FormatPattern 99.9999
      ProcessValue <- "DSE_1_Коэффициент счетчика пасма"
   TextField "Text field_1" at 29,45 size 115x21; Text 'СЧЕТЧИК ПАСМЫ'
   TextField "Text field_2" at 265,45 size 119x21; Text 'СЧЕТЧИК СТРЕНГИ'
   TextField "Text field_3" at 29,65 size 208x20; Text 'Диаметр мерного колеса, мм:'
   TextField "Text field_4" at 29,125 size 154x20; Text 'Импульсов на оборот:'
   TextField "Text field_5" at 29,185 size 82x20; Text 'Коррекция:'
   TextField "Text field_7" at 265,65 size 154x20; Text 'Импульсов на оборот:'
   IOField "I/O field_4" at 271,90 size 96x32; FormatPattern 999.99
      ProcessValue <- "DSE_1_Коэффициент трансмиссии рамки"
   TextField "Text field_8" at 265,125 size 149x20; Text 'Коррекция для шага:'
   IOField "I/O field_5" at 271,150 size 96x32; FormatPattern 99.9999
      ProcessValue <- "DSE_1_Коэффициент метража жилы (выбранной ступени)"
   Button "Button_1" at 378,150 size 38x32; TextOff 'Text'; PictureOff "Graphic_2"
      on Click: ActivateScreen("Settings_2", 0)

screen "Settings_2" 480x272
   Rectangle "Rectangle_9" at 65,60 size 117x40
      Visibility <- "DSE_1_Номер ступени"
   Rectangle "Rectangle_7" at 65,100 size 117x40
      Visibility <- "DSE_1_Номер ступени"
   Rectangle "Rectangle_8" at 65,140 size 117x40
      Visibility <- "DSE_1_Номер ступени"
   Rectangle "Rectangle_6" at 210,220 size 117x40
      Visibility <- "DSE_1_Номер ступени"
   Rectangle "Rectangle_5" at 210,180 size 117x40
      Visibility <- "DSE_1_Номер ступени"
   Rectangle "Rectangle_4" at 210,140 size 117x40
      Visibility <- "DSE_1_Номер ступени"
   Rectangle "Rectangle_10" at 210,100 size 117x40
      Visibility <- "DSE_1_Номер ступени"
   Rectangle "Rectangle_3" at 210,60 size 117x40
      Visibility <- "DSE_1_Номер ступени"
   Rectangle "Rectangle_2" at 65,180 size 117x40
      Visibility <- "DSE_1_Номер ступени"
   Rectangle "Rectangle_1" at 65,220 size 117x40
      Visibility <- "DSE_1_Номер ступени"
   TextField "Text field_6" at 17,5 size 121x30; Text 'настройки'
   Button "Button_3" at 306,7 size 36x28; TextOff 'Text'; PictureOff "NavigateHome_KTP400_Basic_PN_TR"
      on Click: ActivateScreen("DSE1", 0)
   IOField "I/O field_5" at 250,225 size 69x32; FormatPattern 99.9999
      ProcessValue <- "DSE_1_Ступень 9 Коэффициент метража жилы"
   IOField "I/O field_1" at 250,185 size 69x32; FormatPattern 99.9999
      ProcessValue <- "DSE_1_Ступень 8 Коэффициент метража жилы"
   IOField "I/O field_2" at 250,144 size 69x32; FormatPattern 99.9999
      ProcessValue <- "DSE_1_Ступень 7 Коэффициент метража жилы"
   IOField "I/O field_3" at 250,105 size 69x32; FormatPattern 99.9999
      ProcessValue <- "DSE_1_Ступень 6 Коэффициент метража жилы"
   IOField "I/O field_4" at 250,65 size 69x32; FormatPattern 99.9999
      ProcessValue <- "DSE_1_Ступень 5 Коэффициент метража жилы"
   IOField "I/O field_6" at 105,225 size 69x32; FormatPattern 99.9999
      ProcessValue <- "DSE_1_Ступень 4 Коэффициент метража жилы"
   IOField "I/O field_7" at 105,185 size 69x32; FormatPattern 99.9999
      ProcessValue <- "DSE_1_Ступень 3 Коэффициент метража жилы"
   IOField "I/O field_8" at 105,145 size 69x32; FormatPattern 99.9999
      ProcessValue <- "DSE_1_Ступень 2 Коэффициент метража жилы"
   IOField "I/O field_9" at 105,105 size 69x32; FormatPattern 99.9999
      ProcessValue <- "DSE_1_Ступень 1 Коэффициент метража жилы"
   IOField "I/O field_10" at 105,65 size 69x32; FormatPattern 99.9999
      ProcessValue <- "DSE_1_Ступень 0 Коэффициент метража жилы"
   TextField "Text field_9" at 60,65 size 31x29; Text '9'
   TextField "Text field_1" at 65,105 size 31x29; Text '11'
   TextField "Text field_2" at 65,145 size 31x29; Text '14'
   TextField "Text field_3" at 65,185 size 31x29; Text '18'
   TextField "Text field_4" at 65,225 size 31x29; Text '23'
   TextField "Text field_5" at 215,185 size 31x29; Text '63'
   TextField "Text field_7" at 215,145 size 31x29; Text '51'
   TextField "Text field_8" at 215,105 size 31x29; Text '40'
   TextField "Text field_10" at 215,65 size 31x29; Text '32'
   TextField "Text field_11" at 215,225 size 31x29; Text '79'
   TextField "Text field_12" at 17,36 size 354x20; Text 'СЧЕТЧИК СТРЕНГИ: коэфиценты коррекции для шага'
   Button "Button_1" at 20,127 size 32x32; TextOff 'Text'; PictureOff "Left_Arrow"
      on Click: ActivateScreen("DSE1", 0)
   Rectangle "Rectangle_11" at 355,60 size 117x40
      Visibility <- "DSE_1_Номер ступени"
   TextField "Text field_13" at 360,65 size 31x29; Text '91'
   IOField "I/O field_11" at 395,65 size 69x32; FormatPattern 99.9999
      ProcessValue <- "DSE_1_Ступень 10 Коэффициент метража жилы"
*)

(* ===== HMI "HMI_RT_2" =====
system functions are stored by id; their names below are inferred from use
connection "Connection_2": ETHERNET, SMART_S7_1200_OMS
connection "HMI_Connection_2": ETHERNET, SMART_S7_1200_OMS

HMI tags "Default tag table"
   "DSE_1_Метраж пасма" : Real = PLC DSE_3."Метраж пасма", 500 ms
   "DSE_1_метраж жила" : Real = PLC DSE_3."метраж жила", 500 ms
   "DSE_1_Шаг скрутки в метрах (выбранной ступени)" : Real = PLC DSE_3."Шаг скрутки в метрах (выбранной ступени)", 1 s
   "DSE_1_Номер ступени" : Int = PLC DSE_3."Номер ступени", 1 s
   "DSE_1_Сброс счетчика 1" : Bool = PLC DSE_3."Сброс счетчика 1", 1 s
   "DSE_1_Сброс счетчика 2" : Bool = PLC DSE_3."Сброс счетчика 2", 1 s
   "DSE_1_Диаметр колеса пасма" : Real = PLC DSE_3."Диаметр колеса пасма", 1 s
   "DSE_1_Количество импулсов на оборот пасма" : Real = PLC DSE_3."Количество импулсов на оборот пасма", 1 s
   "DSE_1_Коэффициент счетчика пасма" : Real = PLC DSE_3."Коэффициент счетчика пасма", 1 s
   "DSE_1_Коэффициент трансмиссии рамки" : Real = PLC DSE_3."Коэффициент трансмиссии рамки", 1 s
   "DSE_1_Коэффициент метража жилы (выбранной ступени)" : Real = PLC DSE_3."Коэффициент метража жилы (выбранной ступени)", 1 s
   "DSE_1_Метраж заданый" : Real = PLC DSE_3."Метраж заданый", 1 s
   "DSE_1_Ступень 0 Коэффициент метража жилы" : Real = PLC DSE_3."Ступень 0 Коэффициент метража жилы" AT %DB1.DBD0, 1 s
   "DSE_1_Ступень 1 Коэффициент метража жилы" : Real = PLC DSE_3."Ступень 1 Коэффициент метража жилы" AT %DB1.DBD0, 1 s
   "DSE_1_Ступень 2 Коэффициент метража жилы" : Real = PLC DSE_3."Ступень 2 Коэффициент метража жилы" AT %DB1.DBD0, 1 s
   "DSE_1_Ступень 3 Коэффициент метража жилы" : Real = PLC DSE_3."Ступень 3 Коэффициент метража жилы" AT %DB1.DBD0, 1 s
   "DSE_1_Ступень 4 Коэффициент метража жилы" : Real = PLC DSE_3."Ступень 4 Коэффициент метража жилы" AT %DB1.DBD0, 1 s
   "DSE_1_Ступень 5 Коэффициент метража жилы" : Real = PLC DSE_3."Ступень 5 Коэффициент метража жилы" AT %DB1.DBD0, 1 s
   "DSE_1_Ступень 6 Коэффициент метража жилы" : Real = PLC DSE_3."Ступень 6 Коэффициент метража жилы" AT %DB1.DBD0, 1 s
   "DSE_1_Ступень 7 Коэффициент метража жилы" : Real = PLC DSE_3."Ступень 7 Коэффициент метража жилы" AT %DB1.DBD0, 1 s
   "DSE_1_Ступень 8 Коэффициент метража жилы" : Real = PLC DSE_3."Ступень 8 Коэффициент метража жилы" AT %DB1.DBD0, 1 s
   "DSE_1_Ступень 9 Коэффициент метража жилы" : Real = PLC DSE_3."Ступень 9 Коэффициент метража жилы" AT %DB1.DBD0, 1 s
   "DSE_1_Скорость DSE 1" : Real = PLC DSE_3."Скорость DSE 1", 1 s
   "DSE_1_Ступень 10 Коэффициент метража жилы" : Real = PLC DSE_3."Ступень 10 Коэффициент метража жилы" AT %DB1.DBD0, 1 s

text list "Шаг_скрутки": 0 '9'; 1 '11'; 2 '14'; 3 '18'; 4 '23'; 5 '32'; 6 '40'; 7 '51'; 8 '63'; 9 '79'; 10 '91'

screen "DSE3" 480x272, template "Template_1"
   IOField "I/O field_1" at 226,233 size 111x29; FormatPattern 99999.99
      ProcessValue <- "DSE_1_Метраж пасма"
   TextField "Text field_1" at 109,233 size 109x29; Text 'пасма, м:'
   IOField "I/O field_2" at 202,84 size 255x54; FormatPattern 99999.99
      ProcessValue <- "DSE_1_метраж жила"
   TextField "Text field_2" at 7,20 size 113x37; Text 'стренга'
   SymbolicIOField "Symbolic I/O field_1" at 137,52 size 129x37; TextOn '1'; TextOff '0'; TextList "Шаг_скрутки"
      ProcessValue <- "DSE_1_Номер ступени"
   TextField "Text field_5" at 65,63 size 55x29; Text 'шаг:'
   TextField "Text field_3" at 12,101 size 149x29; Text 'намотано, м:'
   IOField "I/O field_3" at 202,177 size 174x41; FormatPattern 99999.9
      ProcessValue <- "DSE_1_Метраж заданый"
   TextField "Text field_4" at 12,179 size 182x29; Text 'установлено, м:'
   TextField "Text field_6" at 218,5 size 76x30; Text 'ДШЁ 3'
   Button "Button_1" at 27,231 size 64x41; TextOff 'сброс'
      on Press: function_b14e0dd5("DSE_1_Сброс счетчика 1", 0)
   Button "Button_2" at 384,231 size 64x41; TextOff 'сброс'
      on Press: function_b14e0dd5("DSE_1_Сброс счетчика 2", 0)
   Button "Button_3" at 428,7 size 37x30; TextOff 'Text'; PictureOff "Graphic_2"; Authorization "User administration"
      on Click: ActivateScreen("Settings", 0)
   TextField "Text field_7" at 12,140 size 188x29; Text 'скорость м/мин:'
   IOField "I/O field_4" at 202,138 size 174x41; FormatPattern 999.9
      ProcessValue <- "DSE_1_Скорость DSE 1"

screen "Settings" 480x272, template "Template_1"
   Button "Button_3" at 306,7 size 36x28; TextOff 'Text'; PictureOff "NavigateHome_KTP400_Basic_PN_TR"
      on Click: ActivateScreen("DSE3", 0)
   TextField "Text field_6" at 17,5 size 248x30; Text 'МАШИНА 1 настройки'
   IOField "I/O field_1" at 35,90 size 96x32; FormatPattern 999.99
      ProcessValue <- "DSE_1_Диаметр колеса пасма"
   IOField "I/O field_2" at 35,150 size 96x32; FormatPattern 99
      ProcessValue <- "DSE_1_Количество импулсов на оборот пасма"
   IOField "I/O field_3" at 35,210 size 96x32; FormatPattern 99.9999
      ProcessValue <- "DSE_1_Коэффициент счетчика пасма"
   TextField "Text field_1" at 29,45 size 115x21; Text 'СЧЕТЧИК ПАСМЫ'
   TextField "Text field_2" at 265,45 size 119x21; Text 'СЧЕТЧИК СТРЕНГИ'
   TextField "Text field_3" at 29,65 size 208x20; Text 'Диаметр мерного колеса, мм:'
   TextField "Text field_4" at 29,125 size 154x20; Text 'Импульсов на оборот:'
   TextField "Text field_5" at 29,185 size 82x20; Text 'Коррекция:'
   TextField "Text field_7" at 265,65 size 154x20; Text 'Импульсов на оборот:'
   IOField "I/O field_4" at 271,90 size 96x32; FormatPattern 999.99
      ProcessValue <- "DSE_1_Коэффициент трансмиссии рамки"
   TextField "Text field_8" at 265,125 size 149x20; Text 'Коррекция для шага:'
   IOField "I/O field_5" at 271,150 size 96x32; FormatPattern 99.9999
      ProcessValue <- "DSE_1_Коэффициент метража жилы (выбранной ступени)"
   Button "Button_1" at 378,150 size 38x32; TextOff 'Text'; PictureOff "Graphic_2"
      on Click: ActivateScreen("Settings_2", 0)

screen "Settings_2" 480x272
   Rectangle "Rectangle_9" at 65,60 size 117x40
      Visibility <- "DSE_1_Номер ступени"
   Rectangle "Rectangle_7" at 65,100 size 117x40
      Visibility <- "DSE_1_Номер ступени"
   Rectangle "Rectangle_8" at 65,140 size 117x40
      Visibility <- "DSE_1_Номер ступени"
   Rectangle "Rectangle_6" at 210,220 size 117x40
      Visibility <- "DSE_1_Номер ступени"
   Rectangle "Rectangle_5" at 210,180 size 117x40
      Visibility <- "DSE_1_Номер ступени"
   Rectangle "Rectangle_4" at 210,140 size 117x40
      Visibility <- "DSE_1_Номер ступени"
   Rectangle "Rectangle_10" at 210,100 size 117x40
      Visibility <- "DSE_1_Номер ступени"
   Rectangle "Rectangle_3" at 210,60 size 117x40
      Visibility <- "DSE_1_Номер ступени"
   Rectangle "Rectangle_2" at 65,180 size 117x40
      Visibility <- "DSE_1_Номер ступени"
   Rectangle "Rectangle_1" at 65,220 size 117x40
      Visibility <- "DSE_1_Номер ступени"
   TextField "Text field_6" at 17,5 size 248x30; Text 'МАШИНА 1 настройки'
   Button "Button_3" at 306,7 size 36x28; TextOff 'Text'; PictureOff "NavigateHome_KTP400_Basic_PN_TR"
      on Click: ActivateScreen("DSE3", 0)
   IOField "I/O field_5" at 250,225 size 69x32; FormatPattern 99.9999
      ProcessValue <- "DSE_1_Ступень 9 Коэффициент метража жилы"
   IOField "I/O field_1" at 250,185 size 69x32; FormatPattern 99.9999
      ProcessValue <- "DSE_1_Ступень 8 Коэффициент метража жилы"
   IOField "I/O field_2" at 250,144 size 69x32; FormatPattern 99.9999
      ProcessValue <- "DSE_1_Ступень 7 Коэффициент метража жилы"
   IOField "I/O field_3" at 250,105 size 69x32; FormatPattern 99.9999
      ProcessValue <- "DSE_1_Ступень 6 Коэффициент метража жилы"
   IOField "I/O field_4" at 250,65 size 69x32; FormatPattern 99.9999
      ProcessValue <- "DSE_1_Ступень 5 Коэффициент метража жилы"
   IOField "I/O field_6" at 105,225 size 69x32; FormatPattern 99.9999
      ProcessValue <- "DSE_1_Ступень 4 Коэффициент метража жилы"
   IOField "I/O field_7" at 105,185 size 69x32; FormatPattern 99.9999
      ProcessValue <- "DSE_1_Ступень 3 Коэффициент метража жилы"
   IOField "I/O field_8" at 105,145 size 69x32; FormatPattern 99.9999
      ProcessValue <- "DSE_1_Ступень 2 Коэффициент метража жилы"
   IOField "I/O field_9" at 105,105 size 69x32; FormatPattern 99.9999
      ProcessValue <- "DSE_1_Ступень 1 Коэффициент метража жилы"
   IOField "I/O field_10" at 105,65 size 69x32; FormatPattern 99.9999
      ProcessValue <- "DSE_1_Ступень 0 Коэффициент метража жилы"
   TextField "Text field_9" at 60,65 size 31x29; Text '9'
   TextField "Text field_1" at 65,105 size 31x29; Text '11'
   TextField "Text field_2" at 65,145 size 31x29; Text '14'
   TextField "Text field_3" at 65,185 size 31x29; Text '18'
   TextField "Text field_4" at 65,225 size 31x29; Text '23'
   TextField "Text field_5" at 215,185 size 31x29; Text '63'
   TextField "Text field_7" at 215,145 size 31x29; Text '51'
   TextField "Text field_8" at 215,105 size 31x29; Text '40'
   TextField "Text field_10" at 215,65 size 31x29; Text '32'
   TextField "Text field_11" at 215,225 size 31x29; Text '79'
   TextField "Text field_12" at 17,36 size 354x20; Text 'СЧЕТЧИК СТРЕНГИ: коэфиценты коррекции для шага'
   Button "Button_1" at 20,127 size 32x32; TextOff 'Text'; PictureOff "Left_Arrow"
      on Click: ActivateScreen("Settings", 0)
   Rectangle "Rectangle_11" at 355,60 size 117x40
      Visibility <- "DSE_1_Номер ступени"
   TextField "Text field_13" at 360,65 size 31x29; Text '91'
   IOField "I/O field_11" at 395,65 size 69x32; FormatPattern 99.9999
      ProcessValue <- "DSE_1_Ступень 10 Коэффициент метража жилы"
*)